// TIA Portal V19 export
DATA_BLOCK "A0301_Trasporto_PERS"   // DB37
// stored: MemoryReserve 100
   VAR RETAIN
      Par : Struct
         Ax { S7_SetPoint := 'True'} : "SpeedMachine_Par";
         Ax_Aut { S7_SetPoint := 'True'} : "A0301_Mach_Speed_Par";
      END_STRUCT;
   END_VAR
BEGIN
   Par.Ax.Man.VelBwd := 10000.0;
   Par.Ax.Man.VelFwdHigh := 10000.0;
   Par.Ax.Man.VelFwdLow := 10000.0;
   Par.Ax.Man.Acc := 1000.0;
   Par.Ax.Man.Dec := 1000.0;
   Par.Ax.Man.DelayChangeVel := T#100MS;
   Par.Ax_Aut.SemiAut_Vel := 15000.0;
   Par.Ax_Aut.Aut_Vel := 20000.0;
   Par.Ax_Aut.Aut_Acc := 1500.0;
   Par.Ax_Aut.Aut_Dec := 1500.0;
END_DATA_BLOCK
